// TIA Portal V21 export
VAR_GLOBAL   // PLC tag table "K_LogoCliente"
END_VAR
VAR_GLOBAL CONSTANT   // user constants
   K_LogoCliente_Brain : Int := 0;
   K_LogoCliente_Jalo : Int := 1;
   K_LogoCliente_Jaloga : Int := 2;
   K_LogoCliente_Greci : Int := 3;
   K_LogoCliente_Sitronic : Int := 4;
   K_LogoCliente_Mutti : Int := 5;
   K_LogoCliente_Casalasco : Int := 6;
   K_LogoCliente_FBL : Int := 7;
   K_LogoCliente_AllGlass : Int := 8;
   K_LogoCliente_Vetromeccanica : Int := 9;
   K_LogoCliente_IngARossi : Int := 10;
   K_LogoCliente_EMS : Int := 11;
   K_LogoCliente_E2Pack : Int := 12;
   K_LogoCliente_Lesaffre : Int := 13;
   K_LogoCliente_Rodolfi : Int := 14;
   K_LogoCliente_Dubit : Int := 15;
END_VAR
